// TwinCAT 3 PLC project PLC
// ProgramVersion: 3.1.4026.19
// CompilerDefines: VISU_USEPROPERTYINFO
// libraries:
//   Tc2_Standard, * (Beckhoff Automation GmbH)
//   Tc2_System, * (Beckhoff Automation GmbH)
//   VisuSymbols, 4.5.0.0 (System)
// project tree:
//   / GlobalTextList.TcGTLO, PlcTask.TcTTO, Visualization Manager.TcVMO (not stored)
//   POUs/ MAIN.TcPOU
//   VISUs/ Visualization.TcVIS

CONFIGURATION PLC
    RESOURCE PLC ON TwinCAT3
        TASK PlcTask(INTERVAL := T#10ms, PRIORITY := 20);
        PROGRAM MAIN WITH PlcTask : MAIN;
    END_RESOURCE
END_CONFIGURATION

// ---- POUs/MAIN.TcPOU
PROGRAM MAIN
VAR
	bStartButton : BOOL; (* Yeşil Başlatma Butonu *)
	bStopButton : BOOL; (* Kırmızı Durdurma Butonu*)
	bMotor : BOOL; (*Çalıştıracağımız Motor*)
END_VAR

IF bStopButton THEN
	bMotor := FALSE;
	
ELSIF bStartButton THEN
	bMotor := TRUE;
END_IF

END_PROGRAM

// ---- VISUs/Visualization.TcVIS
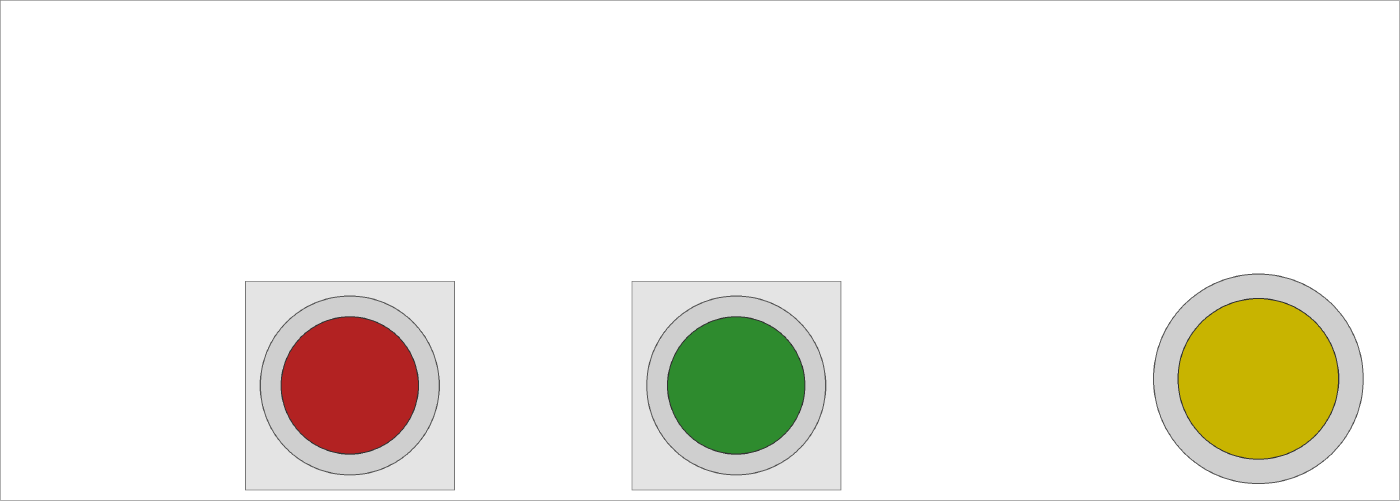
VISUALIZATION Visualization  // 1913x685
    Lamp1 (1526,351 387x334), variable: MAIN.bMotor, style: Lamp-Lamp1-Yellow
    PushSwitch (269,384 418x286), variable: MAIN.bStopButton, behaviour: TOGGLE, style: Switch-PushSwitch-Red
    PushSwitch (797,384 418x286), variable: MAIN.bStartButton, behaviour: TOGGLE, style: Switch-PushSwitch-Green
END_VISUALIZATION
